RoboDK station: Practica_01.rdk

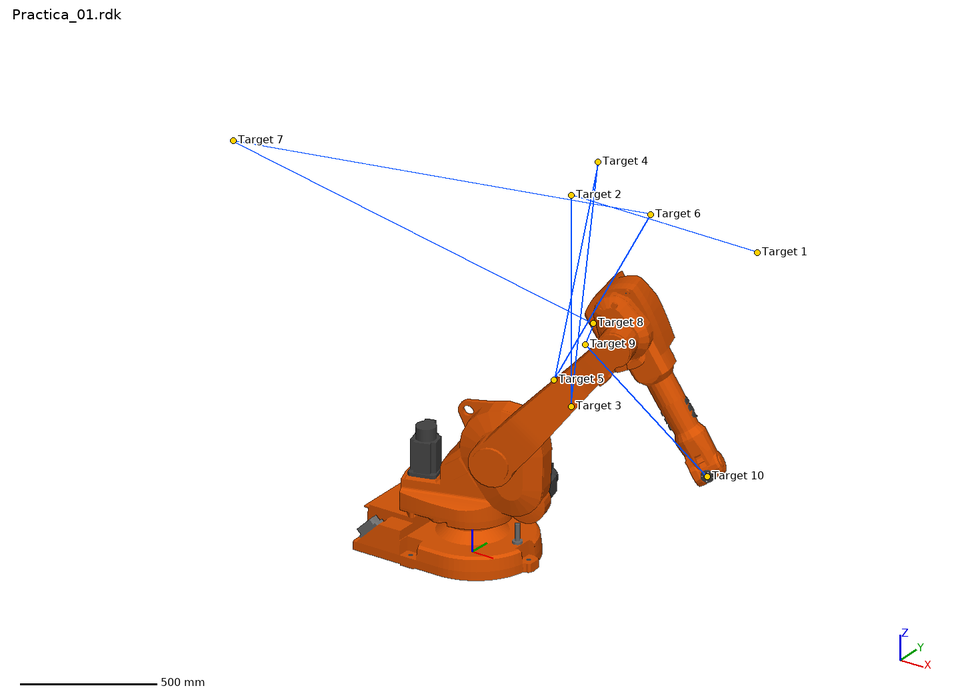
[picture v0: the station drawn from its stored meshes, robots at their saved joint values, targets as dots, program paths as lines]
Station Practica_01 (saved by RoboDK 5.2.1). Poses are relative to the parent item; angles as X-Y-Z fixed-axis rotations.
  - frame ABB IRB 1600-8/1.45 Base at (0, 0, 0) mm
    - robot ABB IRB 1600-8/1.45: 6 axes, payload 8.5 kg, reach 1450 mm, repeatability 0.05 mm, weight 250 kg
        modified DH rows (alpha deg, a mm, theta deg, d mm): 0, 0, 0, 486.5; -90, 150, -90, 0; 0, 700, 0, 0; -90, 0, 0, 600; 90, 0, 0, 0; -90, 0, 180, 65
        joint limits [-180, -90, -245, -200, -115, -400] to [180, 120, 65, 200, 115, 400]; home [0, 0, 0, 0, 0, 0]; saved at [16.257, 41.398, 19.319, 78.311, -73.087, 7.965]
    - target Target 1 (Cartesian target) at (815, 650, 1186.5) mm, rotated rx 0 ry 90 rz 0 deg; joints [40.914, 20.407, -24.606, -85.171, 41.092, 83.604] of ABB IRB 1600-8/1.45
    - target Target 2 (Cartesian target) at (-15, 650, 1186.5) mm, rotated rx 0 ry 90 rz 0 deg; joints [97.017, -7.805, 7.186, -90.076, 97.016, 89.376] of ABB IRB 1600-8/1.45
    - target Target 3 (Cartesian target) at (-15, 650, 326.5) mm, rotated rx 0 ry 90 rz 0 deg; joints [97.017, 51.2, 42.683, -82.999, 89.526, 183.854] of ABB IRB 1600-8/1.45
    - target Target 4 (Cartesian target) at (235, 465, 1466.5) mm, rotated rx 0 ry 90 rz 0 deg; joints [69.918, -14.347, -15.855, -79.579, 72.737, 58.212] of ABB IRB 1600-8/1.45
    - target Target 5 (Cartesian target) at (817.58, -646.62, 1186.54) mm, rotated rx -81.15 ry 90 rz -158.07 deg; joints [-36, 20.4, -24.6, -85.17, 41.09, 83.6] of ABB IRB 1600-8/1.45
    - target Target 6 (Cartesian target) at (726.82, 97.15, 1536.53) mm, rotated rx -81.15 ry 90 rz -158.07 deg; joints [12.698, 8.017, -44.515, -89.769, 89.687, 53.499] of ABB IRB 1600-8/1.45
    - target Target 7 (Cartesian target) at (-875.45, -275.34, 1536.61) mm, rotated rx -81.15 ry 90 rz -158.07 deg; joints [-166.603, 34.277, -86.102, 89.756, 89.808, -38.177] of ABB IRB 1600-8/1.45
    - target Target 8 (Cartesian target) at (550.15, -14.23, 1088.63) mm, rotated rx 69.42 ry 42.73 rz 172.18 deg; joints [-7.83, -14.95, 23.67, 103.17, 105.97, -49.59] of ABB IRB 1600-8/1.45
    - target Target 9 (Cartesian target) at (593.72, -129.43, 1061.51) mm, rotated rx 104.98 ry 52.06 rz 46.56 deg; joints [-7.83, -14.95, 23.67, 94.4, -46.92, -49.59] of ABB IRB 1600-8/1.45
    - target Target 10 (Cartesian target) at (906.61, 200.94, 477.94) mm, rotated rx 104.98 ry 52.06 rz 46.56 deg; joints [16.257, 41.398, 19.319, 78.311, -73.087, 7.965] of ABB IRB 1600-8/1.45
  - program Prog1 (11 instructions, listed below)
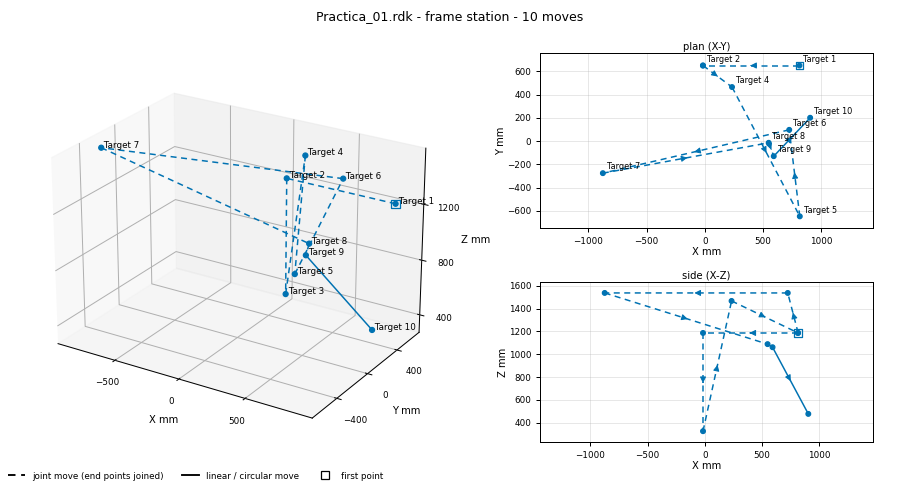
[picture p0: tool path of Practica_01.rdk in frame station, 10 of 10 moves have a stored position in this frame; points joined in program order, loops and branches not executed]

--- program Prog1 (robot ABB IRB 1600-8/1.45) ---
  Est. Ref.: ABB IRB 1600-8/1.45 Base
  MoveJ (Target 1)
  MoveJ (Target 2)
  MoveJ (Target 3)
  MoveJ (Target 4)
  MoveJ (Target 5)
  MoveJ (Target 6)
  MoveJ (Target 7)
  MoveJ (Target 8)
  MoveJ (Target 9)
  MoveL (Target 10)
